TYPE MC_Status :
STRUCT
	
	Status   : BOOL;
	Done   : BOOL;
	Busy   : BOOL;
	Error   : BOOL;
	Active   : BOOL;
	CmdAborted   : BOOL;
	InVelocity   : BOOL;
	ErrorID   : UDINT;
	
	
END_STRUCT
END_TYPE

(* stored: Version 1.1.0.1, ProductVersion 3.1.4024.13
   DUT MC_Status: Id {cc9af087-b4ad-4338-a723-333ea1bd6e50} *)
